Staubli VAL3: ROBERT_TP6_piec.pjx

Parameters version=s7.9 stackSize=5000 millimeterUnit=true
Program file=start.pgx
Program file=stop.pgx
Data file=ROBERT_TP6_piec.dtx
